TYPE PartID : STRING;

END_TYPE

(* stored: Version 1.1.0.1
   DUT PartID: Id {884606e9-013f-465f-9983-af93a481b544} *)
